// TwinCAT 3 PLC project Untitled1
// ProgramVersion: 3.1.4023.0
// libraries:
//   Tc2_Standard, * (Beckhoff Automation GmbH)
//   Tc2_System, * (Beckhoff Automation GmbH)
//   Tc2_TcpIp, * (Beckhoff Automation GmbH)
//   Tc2_Utilities, * (Beckhoff Automation GmbH)
//   Tc3_BA_Common, * (Beckhoff Automation GmbH)
//   Tc3_Module, * (Beckhoff Automation GmbH)
// project tree:
//   DUTs/Types/ DUT.TcDUT (not stored), TcpData.TcDUT (not stored), TcpDataQueue.TcPOU
//   / PlcTask.TcTTO
//   POUs/ MAIN.TcPOU, TcpSingleServerEx.TcPOU
// real-time tasks:
//   TASK PlcTask: cycle T#10ms, priority 20, ADS port 350

CONFIGURATION Untitled1
    RESOURCE PLC ON TwinCAT3
        TASK PlcTask(INTERVAL := T#10ms, PRIORITY := 20);
        PROGRAM MAIN WITH PlcTask : MAIN;
    END_RESOURCE
END_CONFIGURATION

// ---- POUs/MAIN.TcPOU
PROGRAM MAIN
VAR
	visionPC : TcpSingleServerEx;
END_VAR
VAR
	sMessage : STRING := 'from AREA_4';
	newRecipient : STRING;
	
	newData : TcpData;
	retrievedData : TcpData;
	
	sendOnce : BOOL;
	sendFastNum : BOOL;
	
	i : INT := 0;
	
	fbLocalSystemTime : FB_LocalSystemTime;
END_VAR

visionPC(
	ServerNetId:= '', 
	ServerAdr:= , 
	ServerPort:= 8016, 
	busy=> , 
	error=> , 
	errorId=> , 
	bytesReceived=> , 
	receiveStruct=> , 
	connected=> );

IF sendOnce OR sendFastNum THEN
	MEMSET(ADR(newData), 0, SIZEOF(newData));
	
	sMessage := TO_STRING(i);
	
	MEMCPY(ADR(newData), ADR(sMessage), MIN( SIZEOF(newData), SIZEOF(sMessage) ));
	
	IF
		visionPC.queue(data := newData)
	THEN
		i := i + 1;
		sendOnce := FALSE;
	END_IF	
END_IF

END_PROGRAM

// ---- POUs/TcpSingleServerEx.TcPOU
FUNCTION_BLOCK TcpSingleServerEx
VAR_INPUT
	ServerNetId			: STRING; 	(* Server AmsNetId *)
	ServerAdr 			: STRING;	(* Server IP address - IP of the NIC used for this server *)
	ServerPort 			: UDINT := 8016;	(* Server port number *)
END_VAR
VAR_OUTPUT
	busy				: BOOL;
	error				: BOOL;
	errorId				: UDINT;
	bytesReceived		: UDINT;
	
	receiveStruct		: TcpData;	(* Data received *)
	connected 			: BOOL;
END_VAR
VAR
	fbSocketCloseAll 	: FB_SocketCloseAll;
	fbSocketClose 		: FB_SocketClose;
	
	fbSocketListen		: FB_SocketListen;
	fbSocketAccept		: FB_SocketAccept;
	fbSocketReceive		: FB_SocketReceive;
	fbSocketSend 		: FB_SocketSend;
END_VAR
VAR
	listenerSocket		: T_HSOCKET;
	dataSocket			: T_HSOCKET;
END_VAR
VAR
	sendQueue 			: TcpDataQueue;
	sendBuffer 			: ARRAY[0..99] OF BYTE;
	
	sendHeartbeats		: BOOL;
	autoDisconnect		: BOOL;
	
	setupStep 			: (CLOSE_CONNECTIONS, CREATE_LISTENER, ACCEPT_CONNECTION, COMPLETE);
	
	acceptTimer : TON;
	connectionTimer	: TON;
	heartbeatTimer : TON;
END_VAR
VAR_STAT CONSTANT
	connectionTimeout	: TIME := T#30S; //time before connection is closed
	heartbeatInterval	: TIME := T#20S; //heartbeat intervals
	
	incomingHeartbeat	: STRING := 'HEARTBEAT_CLIENT_TO_SERVER';
	outgoingHeartbeat	: STRING := 'HEARTBEAT_SERVER_TO_CLIENT';
END_VAR

blocks();

IF NOT connected THEN
	setup();
END_IF
setupStep := 0;

IF autoDisconnect THEN
	autoDisconnectSeq();
ELSE
	connectionTimer.IN := FALSE;
END_IF

IF sendHeartbeats THEN
	sendHeartbeatSeq();
ELSE
	heartbeatTimer.IN := FALSE;
END_IF

send();
receive(); //receive cyclically

METHOD PRIVATE autoDisconnectSeq : BOOL
connectionTimer(IN := , PT := connectionTimeout, Q => , ET => );
connectionTimer.IN := TRUE;

IF connectionTimer.Q THEN
	connectionTimer.IN := FALSE;
	
	closeSocket(dataSocket);
	//closeSocket(listenerSocket);
	
	setupStep := CLOSE_CONNECTIONS;
	RETURN;
END_IF
END_METHOD

METHOD PRIVATE blocks : BOOL
fbSocketClose(
	sSrvNetId:= ServerNetId, 
	hSocket:= dataSocket, 
	bExecute:= , 
	tTimeout:= , 
	bBusy=> busy, 
	bError=> error, 
	nErrId=> errorId);
	
fbSocketCloseAll(
	sSrvNetId:= ServerNetId, 
	bExecute:= , 
	tTimeout:= , 
	bBusy=> , 
	bError=> , 
	nErrId=> );
(*
IF fbSocketClose.bExecute OR fbSocketCloseAll.bExecute THEN
	fbSocketClose.bExecute := FALSE;
	fbSocketCloseAll.bExecute := FALSE;
END_IF
*)
fbSocketListen(
	sSrvNetId:= ServerNetId, 
	sLocalHost:= ServerAdr, 
	nLocalPort:= ServerPort, 
	bExecute:= , 
	tTimeout:= , 
	bBusy=> busy, 
	bError=> error, 
	nErrId=> errorId, 
	hListener=> listenerSocket);

fbSocketAccept(
	sSrvNetId:= ServerNetId, 
	hListener:= listenerSocket, 
	bExecute:= , 
	tTimeout:= , 
	bAccepted=> , 
	bBusy=> busy, 
	bError=> error, 
	nErrId=> errorId, 
	hSocket=> dataSocket);
	
fbSocketReceive(
	sSrvNetId:= ServerNetId, 
	hSocket:= dataSocket, 
	cbLen:= SIZEOF(receiveStruct), 
	pDest:= ADR(receiveStruct), 
	bExecute:= , 
	tTimeout:= , 
	bBusy=> busy, 
	bError=> error, 
	nErrId=> errorId, 
	nRecBytes=> bytesReceived);
	
fbSocketSend(
	sSrvNetId:= ServerNetId, 
	hSocket:= dataSocket, 
	cbLen:= SIZEOF(sendBuffer), 
	pSrc:= ADR(sendBuffer), 
	bExecute:= , 
	tTimeout:= ,
	bBusy=> busy, 
	bError=> error, 
	nErrId=> errorId);
END_METHOD

METHOD PRIVATE clearBuffer : BOOL
MEMSET(ADR(receiveStruct), 0, SIZEOF(receiveStruct));
END_METHOD

METHOD PRIVATE closeSocket : BOOL
VAR_INPUT
	socket : REFERENCE TO T_HSOCKET;
END_VAR
fbSocketClose.bExecute := TRUE;
fbSocketClose.hSocket := socket;
END_METHOD

METHOD fetch : BOOL
VAR_IN_OUT
	receiverStruct : TcpData;
END_VAR
VAR
	emptyData : TcpData;
END_VAR
fetch := MEMCMP(ADR(receiveStruct), ADR(emptyData), SIZEOF(TcpData)) <> 0; //returns false if no data

receiverStruct := receiveStruct;
receiveStruct := emptyData;
END_METHOD

METHOD queue : BOOL
VAR_INPUT
	data : REFERENCE TO TcpData;
END_VAR
sendQueue.push(data);
END_METHOD

METHOD PRIVATE receive : BOOL
VAR
	heartbeatCheck : STRING;
END_VAR
fbSocketReceive.bExecute := NOT fbSocketReceive.bExecute;
	
MEMCPY(ADR(heartbeatCheck), ADR(receiveStruct), SIZEOF(heartbeatCheck));
IF heartbeatCheck = incomingHeartbeat THEN
	connectionTimer.IN := FALSE;
END_IF
END_METHOD

METHOD PRIVATE send : BOOL
VAR
	polledData : TcpData;
END_VAR
IF NOT fbSocketSend.bBusy THEN
	polledData := sendQueue.poll();
	MEMCPY(ADR(sendBuffer), ADR(polledData), MIN(SIZEOF(polledData), SIZEOF(sendBuffer)));
END_IF

IF NOT BufferIsEmpty(sendBuffer) THEN
	fbSocketSend.bExecute := NOT fbSocketSend.bExecute;
	
ELSE
	fbSocketSend.bExecute := FALSE;
	
END_IF
END_METHOD

METHOD PRIVATE sendHeartbeatSeq : BOOL
VAR
	temp : TcpData;
END_VAR
heartbeatTimer(IN := , PT := heartbeatInterval, Q =>, ET =>);
heartbeatTimer.IN := TRUE;

IF heartbeatTimer.Q THEN
	MEMCPY(ADR(temp), ADR(outgoingHeartbeat), SIZEOF(outgoingHeartbeat));
	queue(temp);
	
	heartbeatTimer.IN := FALSE;
END_IF
END_METHOD

METHOD PRIVATE setup : BOOL
CASE setupStep OF
	CLOSE_CONNECTIONS:
		IF
			fbSocketCloseAll.bExecute AND 
			NOT fbSocketCloseAll.bBusy AND 
			NOT fbSocketCloseAll.bError 
		THEN
			fbSocketCloseAll.bExecute := FALSE;
			setupStep := CREATE_LISTENER;
		ELSE
			fbSocketCloseAll.bExecute := NOT fbSocketCloseAll.bExecute;
		END_IF
		
		//fbSocketCloseAll( bExecute:= TRUE );
		//fbSocketCloseAll( bExecute:= FALSE );
		
	CREATE_LISTENER:
		fbSocketListen.bExecute := TRUE;
		setupStep := ACCEPT_CONNECTION;
		
	ACCEPT_CONNECTION:
		fbSocketListen.bExecute := FALSE;
		
		IF fbSocketListen.bError THEN
			setupStep := CLOSE_CONNECTIONS;
			
		ELSIF NOT fbSocketListen.bBusy THEN
			acceptTimer(IN:= , PT:= T#500MS, Q=> fbSocketAccept.bExecute, ET=> );
			acceptTimer.IN := TRUE;
						
			IF acceptTimer.Q THEN
				acceptTimer.IN := FALSE;
			END_IF
		
			IF fbSocketAccept.bAccepted THEN
				fbSocketAccept.bExecute := FALSE;
				acceptTimer.IN := FALSE;
				setupStep := COMPLETE;
			END_IF
			
		END_IF
		
	COMPLETE:
		connected := TRUE;
		setup := TRUE;
		
END_CASE
END_METHOD

END_FUNCTION_BLOCK

// ---- DUTs/Types/TcpDataQueue.TcPOU
{attribute 'call_after_init'}
FUNCTION_BLOCK TcpDataQueue
VAR
	elements : FB_BA_DynamicArray := (uiEntrySize := SIZEOF(POINTER TO TcpData), uiMinExpCount := CONSTS.initArraySize); 
	length : INT := 0;
	
	entrySize : UDINT;
END_VAR
(*
	this extended version of AdsTcp communication provides the option to dynamically generate ADS messages into a queue
		due to the significant stack memory requirements, the QUEUE model can only be used on systems with adjustable stack
		using QUEUE mode on panel PCs (CP66xx) or other mini controllers can freeze the system
		
	QUEUE mode:
		when a message is polled, a socket with the same recipient name is identified
			if the identified socket is ready to send, then the message is passed to the socket
			otherwise, the message is placed back into the queue
		if no socket with a matching name can be identified, then the message is discarded
		
	SEND mode:
		if a socket matching the recipient name is identified and it is not busy or in error state, then the message is passed
		
	sendMessage() specifies a recipient name and data contents, then checks the mode to determine how to handle the message
*)

METHOD clear : BOOL
VAR
	i : INT;
	temp : REFERENCE TO TcpData;
	tempAdr : POINTER TO TcpData;
END_VAR
FOR i:=0 TO length-1 BY 1 DO
	temp := get(index := i, getSize => );
	tempAdr := ADR(temp);
	__DELETE(tempAdr);
END_FOR

elements.Reset();
length := 0;
END_METHOD

METHOD contains : BOOL //check contents, not pointer value
VAR_INPUT
	value : REFERENCE TO TcpData;
END_VAR
VAR_OUTPUT
	atIndex : INT;
END_VAR
VAR
	temp : REFERENCE TO TcpData;
	i : INT;
END_VAR
IF length = 0 THEN
	contains := FALSE;
	RETURN;
END_IF

FOR i:=0 TO length-1 BY 1 DO
	temp := get(index := i, getSize => );
	
	IF 
		SIZEOF(value) = entrySize AND //same size
		MEMCMP(ADR(temp), ADR(value), SIZEOF(entrySize)) = 0 //same data
	THEN
		contains := TRUE;
		atIndex := i;
		RETURN;
	END_IF
	
END_FOR
contains := FALSE;
END_METHOD

METHOD get : REFERENCE TO TcpData
VAR_INPUT
	index : INT;
END_VAR
VAR_OUTPUT
	getSize : UDINT;
END_VAR
IF length = 0 OR index < 0 OR index >= length THEN
	getSize := 0;
ELSE
	elements.GetEntry(diIndex := index, pResultEntry := ADR(get));
	getSize := SIZEOF(get);
END_IF
END_METHOD

METHOD isEmpty : BOOL
VAR_INPUT
END_VAR
isEmpty := length = 0;
END_METHOD

METHOD poll : TcpData
VAR_OUTPUT
	getSize : UDINT;
END_VAR
IF length > 0 THEN
	poll := get(index := 0, getSize => getSize);
	elements.RemoveEntry(diIndex := 0);
	
	length := length - 1;
END_IF
END_METHOD

METHOD push : BOOL
VAR_INPUT
	value : REFERENCE TO TcpData;
END_VAR
VAR
	temp : POINTER TO TcpData;
END_VAR
temp := __NEW(TcpData);
temp^ := value;

elements.AddEntryPtr(pEntry := temp);

length := length + 1;
END_METHOD

METHOD set : BOOL
VAR_INPUT
	i : INT;
	value : REFERENCE TO TcpData;
END_VAR
VAR
	temp : REFERENCE TO TcpData;
END_VAR
IF length = 0 THEN
	RETURN;
END_IF

IF i >= 0 AND i < length THEN
	temp REF= get(i);
	temp := value;
	
	set := TRUE;
END_IF
END_METHOD

{attribute 'call_after_init'}
METHOD setup : BOOL
VAR_INPUT
END_VAR
entrySize := SIZEOF(TcpData);
END_METHOD

METHOD size : INT
size := length;
END_METHOD

END_FUNCTION_BLOCK
